% RSLogix 500 project test 1111.RSS, saved by version 8.30.00.15 %
PROJECT "UNTITLED"    % processor: MicroLogix 1000 %

PROGRAM FILES
  LAD 2 "MAIN_PROG"  7 rungs
  LAD 3 "USER_FAULT"  1 rungs
  LAD 4 "HSC_INT"  1 rungs
  LAD 5 "STI_INT"  1 rungs
  LAD 6, 7, 8, 9, 10, 11, 12, 13, 14, 15, 16: only END

DATA FILES
  O0 OUTPUT  1 elements
  I1 INPUT  2 elements
  S2 STATUS  33 elements
  B3 BINARY  32 elements
  T4 TIMER  40 elements
  C5 COUNTER  32 elements
  R6 CONTROL  16 elements
  N7 INTEGER  105 elements

LADDER 2 "MAIN_PROG"
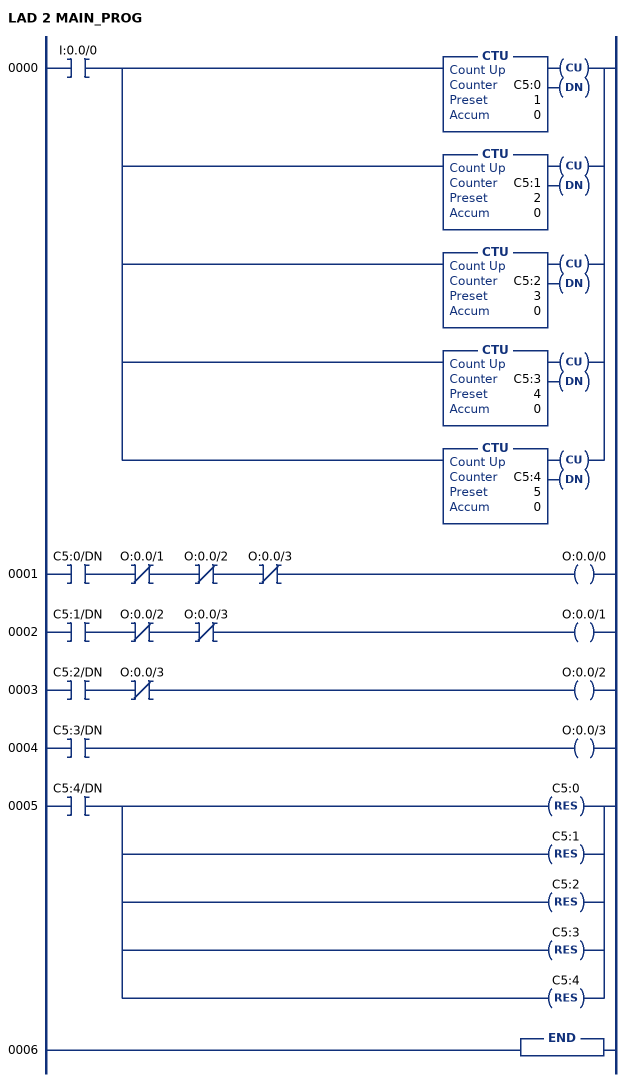
% Rung: 0 %
SOR XIC I:0.0/0 BST BST BST BST CTU C5:0 1 0 NXB CTU C5:1 2 0 BND NXB CTU C5:2 3 0 BND NXB CTU C5:3 4 0 BND NXB CTU C5:4 5 0 BND EOR
% Rung: 1 %
SOR XIC C5:0/DN XIO O:0.0/1 XIO O:0.0/2 XIO O:0.0/3 OTE O:0.0/0 EOR
% Rung: 2 %
SOR XIC C5:1/DN XIO O:0.0/2 XIO O:0.0/3 OTE O:0.0/1 EOR
% Rung: 3 %
SOR XIC C5:2/DN XIO O:0.0/3 OTE O:0.0/2 EOR
% Rung: 4 %
SOR XIC C5:3/DN OTE O:0.0/3 EOR
% Rung: 5 %
SOR XIC C5:4/DN BST BST BST BST RES C5:0 NXB RES C5:1 BND NXB RES C5:2 BND NXB RES C5:3 BND NXB RES C5:4 BND EOR
% Rung: 6 %
SOR END EOR

DATA TABLE (non-zero values as saved)
DATA C5
% .PRE .ACC %
% C5:0 % 1 0
% C5:1 % 2 0
% C5:2 % 3 0
% C5:3 % 4 0
% C5:4 % 5 0
